(* Schneider Machine Expert - Basic project Seren1, file version 3.0.0.0 *)

HARDWARE
  Cpu 0: TM221CE16R
  EthernetConfiguration: NetworkName=M221, IpAllocationMode=FixedAddress, IpAddress=192.168.0.221, SubnetMask=255.255.255.0
  SerialLineConfiguration: Baud=Baud19200, Parity=ParityEven, DataBits=DataBits8, StopBits=StopBits1, PhysicalMedium=PhysicalMediumRs485, TransmissionMode=TransmissionModeModbusRtu, SlaveId=1, Addressing=SlaveAddressing
  MastTask: UsePeriodScanMode=false, PeriodScan=100
  FastTask: Period=255
  CpuBehavior: StartingMode=StartInRun, AutoSaveRamOnEeprom=true, WatchdogPeriod=250

SYMBOLS  (address, symbol, comment, settings)
  %MW0      PLC_CONTROL_WORD
  %MW1      PLC_STATUS_WORD
  %MW2      ALLERT_1_COUNT
  %MW3      ALLERT_1_PERIOD
  %MW4      ALLERT_1_CICLE
  %TM0        [Preset=1, Base=OneSecond]
  %TM1        [Preset=1, Base=OneSecond]
  %TM2        [Preset=5, Base=OneHundredMilliSeconds]
  %TM3        [Preset=5, Base=OneHundredMilliSeconds]
  %QWM0     QW_HEARD_BEAT_WORD
  %QWM1     QW_PLC_CONTROL_WORD
  %IWM0     IW_PLC_HEARD_BEAT_WORD
  %IWM1     IW_PLC_STATUS_WORD

POU New POU
  (* SectionNumber=1 *)

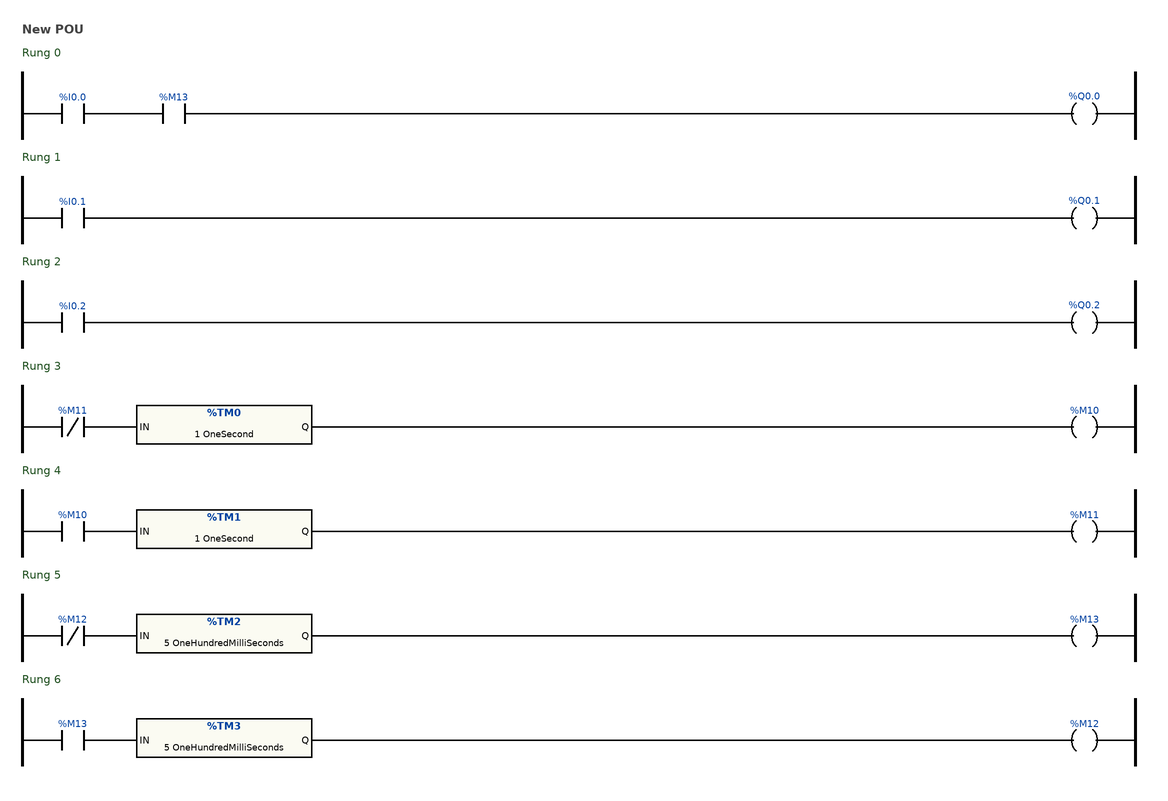

// Rung 0
  LD %I0.0
  AND %M13
  ST %Q0.0
  // as ST:
  //   %Q0.0 := %I0.0 AND %M13;

// Rung 1
  LD %I0.1
  ST %Q0.1
  // as ST:
  //   %Q0.1 := %I0.1;

// Rung 2
  LD %I0.2
  ST %Q0.2
  // as ST:
  //   %Q0.2 := %I0.2;

// Rung 3
  BLK %TM0
  LDN %M11
  IN
  OUT_BLK
  LD Q
  ST %M10
  END_BLK
  // as ST:
  //   %TM0(IN := NOT %M11);
  //   %M10 := %TM0.Q;

// Rung 4
  BLK %TM1
  LD %M10
  IN
  OUT_BLK
  LD Q
  ST %M11
  END_BLK
  // as ST:
  //   %TM1(IN := %M10);
  //   %M11 := %TM1.Q;

// Rung 5
  BLK %TM2
  LDN %M12
  IN
  OUT_BLK
  LD Q
  ST %M13
  END_BLK
  // as ST:
  //   %TM2(IN := NOT %M12);
  //   %M13 := %TM2.Q;

// Rung 6
  BLK %TM3
  LD %M13
  IN
  OUT_BLK
  LD Q
  ST %M12
  END_BLK
  // as ST:
  //   %TM3(IN := %M13);
  //   %M12 := %TM3.Q;

POU ModBusExchange
  (* SectionNumber=2 *)

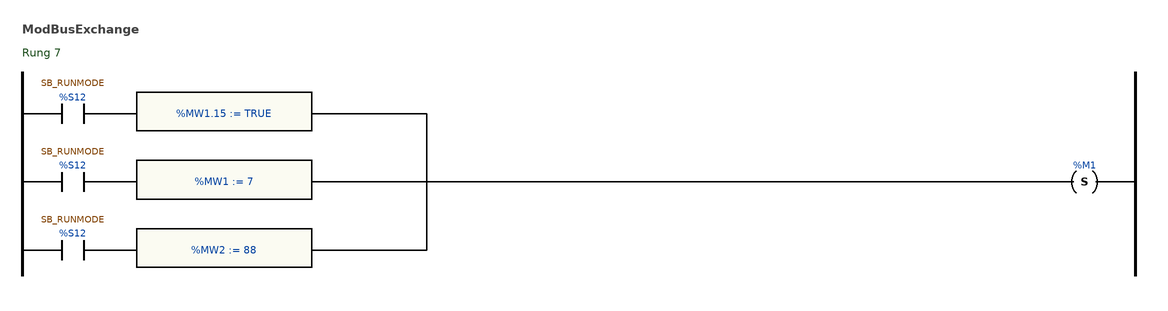

// Rung 7
  // %S12: The controller is running
  (* no IL stored for this rung *)
